// Mitsubishi GX Works2 project: Project 0   PLC: Q03UDV

PROGRAM MAIN
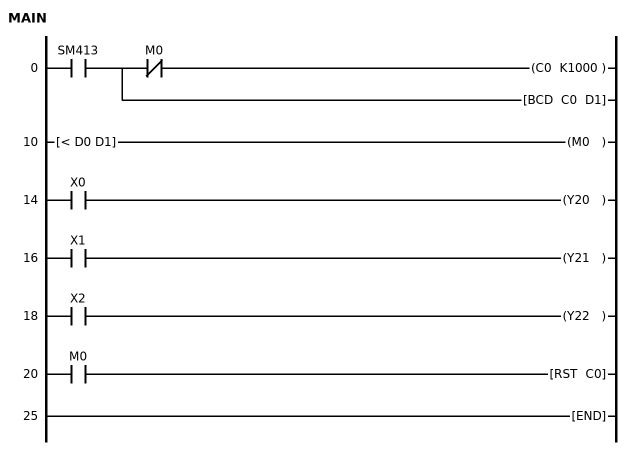
0     LD      SM413
      MPS
      ANI     M0
      OUT     C0 K1000
      MPP
      BCD     C0 D1
10    LD<     D0 D1
      OUT     M0
14    LD      X0
      OUT     Y20
16    LD      X1
      OUT     Y21
18    LD      X2
      OUT     Y22
20    LD      M0
      RST     C0
25    END
END_PROGRAM
